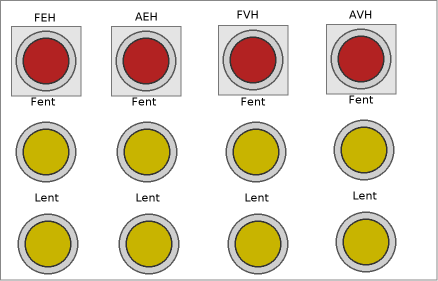
VISUALIZATION TempJozsiHajlitok  // 438x281
    PushSwitch (11,26 70x70), variable: HAJLITOK.bElohajlitoFelso, behaviour: TOGGLE, style: Switch-PushSwitch-Red
    Label (11,3 68x30), "FEH"
    PushSwitch (111,26 70x70), variable: HAJLITOK.bElohajlitoAlso, behaviour: TOGGLE, style: Switch-PushSwitch-Red
    Label (118,2 57x30), "AEH"
    PushSwitch (218,25 70x70), variable: HAJLITOK.bVeghajlitoFelso, behaviour: TOGGLE, style: Switch-PushSwitch-Red
    Label (173,0 150x30), "FVH"
    PushSwitch (326,24 70x70), variable: HAJLITOK.bVeghajlitoAlso, behaviour: TOGGLE, style: Switch-PushSwitch-Red
    Label (286,0 150x30), "AVH"
    Lamp1 (13,209 70x70), variable: HAJLITOK.bElohajlitoFelsoLent, style: Lamp-Lamp1-Yellow
    Label (-8,183 110x30), "Lent"
    Lamp1 (11,117 70x70), variable: HAJLITOK.bElohajlitoFelsoFent, style: Lamp-Lamp1-Yellow
    Label (-12,87 110x30), "Fent"
    Lamp1 (114,209 70x70), variable: HAJLITOK.bElohajlitoAlsoLent, style: Lamp-Lamp1-Yellow
    Label (93,183 110x30), "Lent"
    Lamp1 (112,117 70x70), variable: HAJLITOK.bElohajlitoAlsoFent, style: Lamp-Lamp1-Yellow
    Label (89,87 110x30), "Fent"
    Lamp1 (223,209 70x70), variable: HAJLITOK.bVeghajlitoFelsoLent, style: Lamp-Lamp1-Yellow
    Label (202,183 110x30), "Lent"
    Lamp1 (221,117 70x70), variable: HAJLITOK.bVeghajlitoFelsoFent, style: Lamp-Lamp1-Yellow
    Label (198,87 110x30), "Fent"
    Lamp1 (331,207 70x70), variable: HAJLITOK.bVeghajlitoAlsoLent, style: Lamp-Lamp1-Yellow
    Label (310,181 110x30), "Lent"
    Lamp1 (329,115 70x70), variable: HAJLITOK.bVeghajlitoAlsoFent, style: Lamp-Lamp1-Yellow
    Label (306,85 110x30), "Fent"
END_VISUALIZATION

(* stored: Version 1.1.0.1, ProductVersion 3.1.4024.11
   Visu TempJozsiHajlitok: Id {32665308-b384-4ae0-8594-f8c0382b26fb} *)
